// TIA Portal V16 export
// export: Created 2021-12-01T20:36:11.8852293Z, ExportSetting WithDefaults, DisplayName Totally Integrated Automation Portal, DisplayVersion V16 Update 4, DisplayName TIA Portal Version Control Interface, DisplayVersion V16 Update 2, DisplayName TIA Portal Openness, DisplayVersion V16 Update 4, DisplayName SINAMICS Startdrive Advanced, DisplayVersion V16 Update 5, DisplayName SINAMICS Startdrive G130, G150, S120, S150, SINAMICS MV, S210, DisplayVersion V16 Update 5, DisplayName SINAMICS Startdrive G110M, G120, G120C, G120D, G120P, G115D, DisplayVersion V16 Update 5, DisplayName STEP 7 Professional, DisplayVersion V16 Update 4, DisplayName STEP 7 Safety, DisplayVersion V16, DisplayName WinCC Advanced, DisplayVersion V16 Update 4
DATA_BLOCK "ST00310_FX01_VFD01_IDB"   // DB77
AUTHOR : Tesla
FAMILY : Drive
VERSION : 1.0
// stored: AssignedProDiagFB OPMODE02_PD, AutoNumber false, DBAccessibleFromOPCUA true, InstanceOfName DRIVE_SEW_3PIO_PD_FB, InstanceOfType FB
"DRIVE_SEW_3PIO_PD_FB"
   // VAR_INPUT
   //    PLANT_IDENTIFIER { ExternalAccessible := 'False'; ExternalVisible := 'False'; ExternalWritable := 'False'} : WString[24];
   //    HARDWARE_OK { ExternalAccessible := 'False'; ExternalVisible := 'False'; ExternalWritable := 'False'} : Bool;
   //    SAFETY_OK { ExternalAccessible := 'False'; ExternalVisible := 'False'; ExternalWritable := 'False'} : Bool;
   //    HW_ID { ExternalAccessible := 'False'; ExternalVisible := 'False'; ExternalWritable := 'False'} : HW_IO;
   //    HEADUNIT_HW_ID { ExternalAccessible := 'False'; ExternalVisible := 'False'; ExternalWritable := 'False'} : HW_IO;
   //    SET_PARAMETER_2 { ExternalAccessible := 'False'; ExternalVisible := 'False'; ExternalWritable := 'False'} : Bool;
   //    CLOCKWISE_ROTATION { ExternalAccessible := 'False'; ExternalVisible := 'False'; ExternalWritable := 'False'} : Bool;
   //    COUNTERCLOCKWISE_ROTATION { ExternalAccessible := 'False'; ExternalVisible := 'False'; ExternalWritable := 'False'} : Bool;
   //    DIR_INDICATOR { ExternalAccessible := 'False'; ExternalVisible := 'False'; ExternalWritable := 'False'} : Bool;
   //    HIDE_ALARM_ALL { ExternalAccessible := 'False'; ExternalVisible := 'False'; ExternalWritable := 'False'} : Bool;
   //    FAST_SPEED { ExternalAccessible := 'False'; ExternalVisible := 'False'; ExternalWritable := 'False'} : Bool;
   //    VALUE_FAST_SPEED { ExternalAccessible := 'False'; ExternalVisible := 'False'; ExternalWritable := 'False'} : Real;
   //    SLOW_SPEED { ExternalAccessible := 'False'; ExternalVisible := 'False'; ExternalWritable := 'False'} : Bool;
   //    VALUE_SLOW_SPEED { ExternalAccessible := 'False'; ExternalVisible := 'False'; ExternalWritable := 'False'} : Real;
   //    JOG_SPEED { ExternalAccessible := 'False'; ExternalVisible := 'False'; ExternalWritable := 'False'} : Bool;
   //    VALUE_JOG_SPEED { ExternalAccessible := 'False'; ExternalVisible := 'False'; ExternalWritable := 'False'} : Real;
   //    RAPID_STOP { ExternalAccessible := 'False'; ExternalVisible := 'False'; ExternalWritable := 'False'} : Bool;
   //    RESET { ExternalAccessible := 'False'; ExternalVisible := 'False'; ExternalWritable := 'False'} : Bool;
   //    SPEED_DISPLAY_MODE { ExternalAccessible := 'False'; ExternalVisible := 'False'; ExternalWritable := 'False'} : Int;
   //    MECHNICAL_FACTOR { ExternalAccessible := 'False'; ExternalVisible := 'False'; ExternalWritable := 'False'} : Real;
   //    OPEN_BRAKE { ExternalAccessible := 'False'; ExternalVisible := 'False'; ExternalWritable := 'False'} : Bool;
   //    VALUE_RAMP_UP { ExternalAccessible := 'False'; ExternalVisible := 'False'; ExternalWritable := 'False'} : Int;
   //    VALUE_RAMP_DOWN { ExternalAccessible := 'False'; ExternalVisible := 'False'; ExternalWritable := 'False'} : Int;
   // END_VAR
   // VAR_OUTPUT
   //    GENERAL_ALARM { ExternalAccessible := 'False'; ExternalVisible := 'False'; ExternalWritable := 'False'} : Bool;
   //    OUTPUT_STAGE_ENABLED { ExternalAccessible := 'False'; ExternalVisible := 'False'; ExternalWritable := 'False'} : Bool;
   //    INVERTER_READY { ExternalAccessible := 'False'; ExternalVisible := 'False'; ExternalWritable := 'False'} : Bool;
   //    DRIVE_READY { ExternalAccessible := 'False'; ExternalVisible := 'False'; ExternalWritable := 'False'} : Bool;
   //    DRIVE_RUNNING { ExternalAccessible := 'False'; ExternalVisible := 'False'; ExternalWritable := 'False'} : Bool;
   //    PARAMETER_2_SET { ExternalAccessible := 'False'; ExternalVisible := 'False'; ExternalWritable := 'False'} : Bool;
   // END_VAR
   // VAR_IN_OUT
   //    IF_HMI : "DRIVE_SEW_HMI_UDT";
   // END_VAR
   // VAR
   //    DataExchangeReceive { ExternalAccessible := 'False'; ExternalVisible := 'False'; ExternalWritable := 'False'} : "DRIVE_SEW_3PIO_SPEED_RECV_UDT";
   //    DataExchangeSend { ExternalAccessible := 'False'; ExternalVisible := 'False'; ExternalWritable := 'False'} : "DRIVE_SEW_3PIO_SPEED_SEND_UDT";
   //    Instruction { ExternalAccessible := 'False'; ExternalVisible := 'False'; ExternalWritable := 'False'} : Struct
   //       Timer_AlarmDelay { ExternalAccessible := 'False'; ExternalVisible := 'False'; ExternalWritable := 'False'} : IEC_TIMER;
   //    END_STRUCT;
   //    AX { ExternalAccessible := 'False'; ExternalVisible := 'False'; ExternalWritable := 'False'} : Struct
   //       General_Alarm { ExternalAccessible := 'False'; ExternalVisible := 'False'; ExternalWritable := 'False'} : Bool;
   //       DriveReady { ExternalAccessible := 'False'; ExternalVisible := 'False'; ExternalWritable := 'False'} : Bool;
   //       "24VOperation" { ExternalAccessible := 'False'; ExternalVisible := 'False'; ExternalWritable := 'False'} : Bool;
   //       ControlInhibit { ExternalAccessible := 'False'; ExternalVisible := 'False'; ExternalWritable := 'False'} : Bool;
   //       NoEnable { ExternalAccessible := 'False'; ExternalVisible := 'False'; ExternalWritable := 'False'} : Bool;
   //       StandstillCur { ExternalAccessible := 'False'; ExternalVisible := 'False'; ExternalWritable := 'False'} : Bool;
   //       Enable { ExternalAccessible := 'False'; ExternalVisible := 'False'; ExternalWritable := 'False'} : Bool;
   //       ManuOpEn { ExternalAccessible := 'False'; ExternalVisible := 'False'; ExternalWritable := 'False'} : Bool;
   //       EnableRight { ExternalAccessible := 'False'; ExternalVisible := 'False'; ExternalWritable := 'False'} : Bool;
   //       EnableLeft { ExternalAccessible := 'False'; ExternalVisible := 'False'; ExternalWritable := 'False'} : Bool;
   //       HideAlarmDelay { ExternalAccessible := 'False'; ExternalVisible := 'False'; ExternalWritable := 'False'} : Bool;
   //       AlarmPD_NoChange { ExternalAccessible := 'False'; ExternalVisible := 'False'; ExternalWritable := 'False'} : Bool;
   //       Last_AlarmNoPD { ExternalAccessible := 'False'; ExternalVisible := 'False'; ExternalWritable := 'False'} : UInt;
   //       ENBlock { ExternalAccessible := 'False'; ExternalVisible := 'False'; ExternalWritable := 'False'; S7_SetPoint := 'True'} : IEC_TIMER;
   //       HideAlarmTimer { ExternalAccessible := 'False'; ExternalVisible := 'False'; ExternalWritable := 'False'; S7_SetPoint := 'True'} : IEC_TIMER;
   //    END_STRUCT;
   //    PE { ExternalAccessible := 'False'; ExternalVisible := 'False'; ExternalWritable := 'False'} : Struct
   //       Reset { ExternalAccessible := 'False'; ExternalVisible := 'False'; ExternalWritable := 'False'} : Bool;
   //       ParaChange { ExternalAccessible := 'False'; ExternalVisible := 'False'; ExternalWritable := 'False'} : Bool;
   //       Alarm_Change { ExternalAccessible := 'False'; ExternalVisible := 'False'; ExternalWritable := 'False'} : Bool;
   //       Alarm_Incoming { ExternalAccessible := 'False'; ExternalVisible := 'False'; ExternalWritable := 'False'} : Bool;
   //    END_STRUCT;
   //    PP { ExternalAccessible := 'False'; ExternalVisible := 'False'; ExternalWritable := 'False'} : Struct
   //       Reset { ExternalAccessible := 'False'; ExternalVisible := 'False'; ExternalWritable := 'False'} : Bool;
   //       ParaChange { ExternalAccessible := 'False'; ExternalVisible := 'False'; ExternalWritable := 'False'} : Bool;
   //       Alarm_Change { ExternalAccessible := 'False'; ExternalVisible := 'False'; ExternalWritable := 'False'} : Bool;
   //       Alarm_Incoming { ExternalAccessible := 'False'; ExternalVisible := 'False'; ExternalWritable := 'False'} : Bool;
   //    END_STRUCT;
   //    NE { ExternalAccessible := 'False'; ExternalVisible := 'False'; ExternalWritable := 'False'} : Struct
   //       Reset { ExternalAccessible := 'False'; ExternalVisible := 'False'; ExternalWritable := 'False'} : Bool;
   //       ParaChange { ExternalAccessible := 'False'; ExternalVisible := 'False'; ExternalWritable := 'False'} : Bool;
   //    END_STRUCT;
   //    NP { ExternalAccessible := 'False'; ExternalVisible := 'False'; ExternalWritable := 'False'} : Struct
   //       Reset { ExternalAccessible := 'False'; ExternalVisible := 'False'; ExternalWritable := 'False'} : Bool;
   //       ParaChange { ExternalAccessible := 'False'; ExternalVisible := 'False'; ExternalWritable := 'False'} : Bool;
   //    END_STRUCT;
   //    wrk { ExternalAccessible := 'False'; ExternalVisible := 'False'; ExternalWritable := 'False'} : Struct
   //       FaultCode { ExternalAccessible := 'False'; ExternalVisible := 'False'; ExternalWritable := 'False'} : Int;
   //       UnitStatusCode { ExternalAccessible := 'False'; ExternalVisible := 'False'; ExternalWritable := 'False'} : Int;
   //    END_STRUCT;
   //    HardwareFault { ExternalAccessible := 'False'; ExternalVisible := 'False'; ExternalWritable := 'False'} : Bool;
   //    MainSwitchOff { ExternalAccessible := 'False'; ExternalVisible := 'False'; ExternalWritable := 'False'} : Bool;
   //    AlarmActive { ExternalAccessible := 'False'; ExternalVisible := 'False'; ExternalWritable := 'False'} : Bool;
   //    ConvActualSpeed { ExternalAccessible := 'False'; ExternalVisible := 'False'; ExternalWritable := 'False'} : Real;
   //    ConvActualCurrent { ExternalAccessible := 'False'; ExternalVisible := 'False'; ExternalWritable := 'False'} : Int;
   //    SpeedSetPoint_selected { ExternalAccessible := 'False'; ExternalVisible := 'False'; ExternalWritable := 'False'} : Real;
   //    Comm_OK { ExternalAccessible := 'False'; ExternalVisible := 'False'; ExternalWritable := 'False'} : Bool;
   //    Alarm_No_PD { ExternalAccessible := 'False'; ExternalVisible := 'False'; ExternalWritable := 'False'} : UInt;
   //    GLOBAL_TECUNIT_AlarmTextList_Item { ExternalAccessible := 'False'; ExternalVisible := 'False'; ExternalWritable := 'False'} : USInt;
   //    GLOBAL_TECUNIT_WarningTextList_Item { ExternalAccessible := 'False'; ExternalVisible := 'False'; ExternalWritable := 'False'} : USInt;
   //    Warning_No_PD { ExternalAccessible := 'False'; ExternalVisible := 'False'; ExternalWritable := 'False'} : Array[1..9] of USInt;
   // END_VAR
BEGIN
END_DATA_BLOCK
